FUNCTION_BLOCK FB_StationT1
VAR_IN_OUT
	XpMover			: MC_PlanarMover;
	XpTrack			: ARRAY[*] OF MC_PlanarTrack;
END_VAR
VAR_INPUT
	execute			: BOOL;
	bT2Ready		: BOOL :=TRUE;
	bT3Ready		: BOOL :=TRUE;
END_VAR
VAR_OUTPUT
	bOccupied		: BOOL;
	bReady			: BOOL;
	bDone			: BOOL;
END_VAR
VAR
	nState			: INT;
	fbMoveTrack		: FB_XpMoveTrack;
	nTargetTrack	: INT;
	bMove			: BOOL;
END_VAR

CASE nState OF
	0://init
	IF execute THEN
		bOccupied := TRUE;//Stationの状態をOccupiedにする
		bReady := FALSE;
		bDone	:= FALSE;
		nState := 10;
	END_IF
	
	10://判断
	IF bT2Ready THEN
		nTargetTrack := E_TrackName.T2_1_ToLink;//右ルート
		nState := 20;
	ELSIF bT3Ready THEN
		nTargetTrack := E_TrackName.T3_1_ToLink;//左ルート
		nState := 20;
	END_IF
	
	20://移動
	IF XpMover.MCTOPLC.SETONTRACK.SetVelo=0 THEN
		bMove := TRUE;
		fbMoveTrack.execute := TRUE;
		nState := 30;
	END_IF
	
	30:
	IF fbMoveTrack.done THEN
		fbMoveTrack.execute := FALSE;
		bOccupied := FALSE;
		bReady := TRUE;
		bMove := FALSE;
		bDone := TRUE;
		nState := 40;
	END_IF
	
	40://initへ戻る
	nState := 0;
END_CASE

fbMoveTrack(XpMover:= XpMover, 
		XpTrack:= XpTrack[nTargetTrack]);

END_FUNCTION_BLOCK

(* stored: Version 1.1.0.1
   POU FB_StationT1: Id {ce1d8752-903b-4abe-8510-95224edda60b}, SpecialFunc None *)
